FUNCTION_BLOCK fb_prod_feedforward
VAR_INPUT
END_VAR
VAR_OUTPUT
END_VAR
VAR
END_VAR

END_FUNCTION_BLOCK

(* stored: Version 1.1.0.1, ProductVersion 3.1.0.26
   POU fb_prod_feedforward: Id {96b2eeae-4de0-4c6e-85db-c90a80da890a} *)
